// TIA Portal V18 program export: 0 tag tables, 0 data types, 0 data blocks, 3 code blocks (in call order from the OBs), 0 instance data blocks

ORGANIZATION_BLOCK "Main"   // OB1, LAD, ProgramCycle
TITLE = "Main Program Sweep (Cycle)"
{ S7_Optimized_Access := 'TRUE' }
// stored: SetENOAutomatically false
   VAR_INPUT
      Initial_Call : Bool;
      Remanence : Bool;
   END_VAR
BEGIN
END_ORGANIZATION_BLOCK

FUNCTION_BLOCK "Baustein_1"   // FB1, FBD
{ S7_Optimized_Access := 'TRUE' }
// stored: MemoryReserve 100, SetENOAutomatically false
   VAR_OUTPUT
      Input_1 : Bool;
      Input_2 : Int := 200;
      Input_3 : Int := 2001;
   END_VAR
BEGIN

REGION Network 1
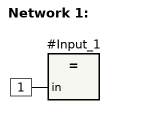
   #Input_1 := 1;
END_REGION
END_FUNCTION_BLOCK

FUNCTION_BLOCK "Baustein_Int"   // FB2, FBD
{ S7_Optimized_Access := 'TRUE' }
// stored: MemoryReserve 100, SetENOAutomatically false
   VAR_INPUT
      Test_1 : Int := 120;
      Test_2 : Bool := true;
   END_VAR
   VAR_OUTPUT
      Output_1 : Int := 120;
      Output_2_1 : Int := 78;
      Output_2 : Bool := true;
   END_VAR
BEGIN
END_FUNCTION_BLOCK
